SYSTEM Demo
  (* Version 1.0, 2022-05-14, Maximilian Scharf *)
  APPLICATION DemoApp
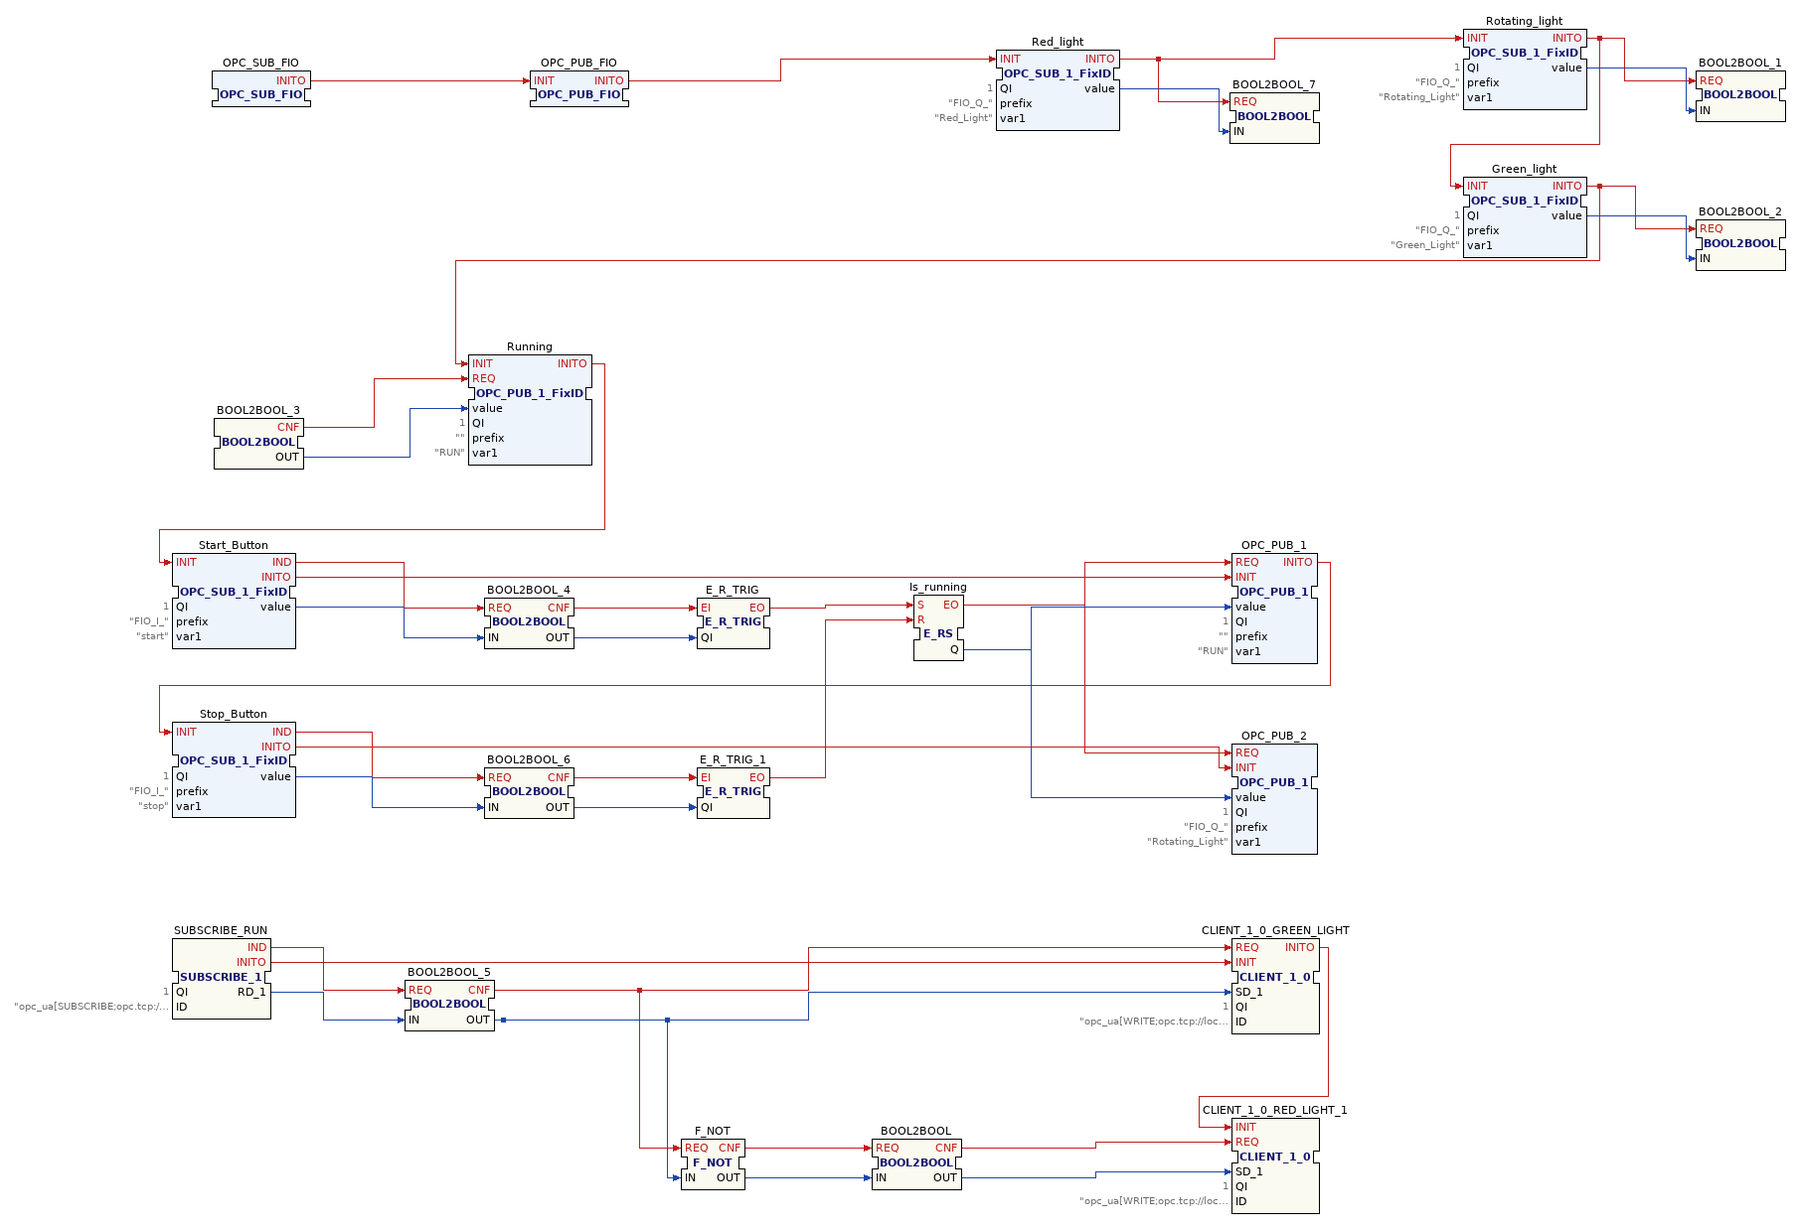
    (* Group __Group01: Factory IO controlpanel *)
    (* Group __Group02: Create nodes on server, which are used on clients *)
    (* Group __Group03: node RUN only writeable for server-forte *)
    FBS
      BOOL2BOOL_1 : BOOL2BOOL; {SET_ATTRIBUTE(GroupName, __Group02)}
      BOOL2BOOL_2 : BOOL2BOOL; {SET_ATTRIBUTE(GroupName, __Group02)}
      BOOL2BOOL_4 : BOOL2BOOL;
      Is_running : E_RS;
      BOOL2BOOL_5 : BOOL2BOOL;
      SUBSCRIBE_RUN : SUBSCRIBE_1(QI := 1, ID := "opc_ua[SUBSCRIBE;opc.tcp://localhost:4840#;/Objects/RUN]");
      CLIENT_1_0_GREEN_LIGHT : CLIENT_1_0(QI := 1, ID := "opc_ua[WRITE;opc.tcp://localhost:4840#;/Objects/FIO_Q_Green_Light]");
      BOOL2BOOL_3 : BOOL2BOOL; {SET_ATTRIBUTE(GroupName, __Group03)}
      E_R_TRIG : E_R_TRIG;
      E_R_TRIG_1 : E_R_TRIG;
      BOOL2BOOL_6 : BOOL2BOOL;
      BOOL2BOOL_7 : BOOL2BOOL; {SET_ATTRIBUTE(GroupName, __Group02)}
      F_NOT : F_NOT;
      CLIENT_1_0_RED_LIGHT_1 : CLIENT_1_0(QI := 1, ID := "opc_ua[WRITE;opc.tcp://localhost:4840#;/Objects/FIO_Q_Red_Light]");
      BOOL2BOOL : BOOL2BOOL;
    END_FBS
    SUBAPPS
      OPC_PUB_FIO : OPC_PUB_FIO; {SET_ATTRIBUTE(GroupName, __Group01)}
      Start_Button : OPC_SUB_1_FixID(QI := 1, prefix := "FIO_I_", var1 := "start");
      Rotating_light : OPC_SUB_1_FixID(QI := 1, prefix := "FIO_Q_", var1 := "Rotating_Light"); {SET_ATTRIBUTE(GroupName, __Group02)}
      Green_light : OPC_SUB_1_FixID(QI := 1, prefix := "FIO_Q_", var1 := "Green_Light"); {SET_ATTRIBUTE(GroupName, __Group02)}
      OPC_SUB_FIO : OPC_SUB_FIO; {SET_ATTRIBUTE(GroupName, __Group01)}
      OPC_PUB_1 : OPC_PUB_1(QI := 1, prefix := "", var1 := "RUN");
      OPC_PUB_2 : OPC_PUB_1(QI := 1, prefix := "FIO_Q_", var1 := "Rotating_Light");
      Running : OPC_PUB_1_FixID(QI := 1, prefix := "", var1 := "RUN"); {SET_ATTRIBUTE(GroupName, __Group03)}
      Stop_Button : OPC_SUB_1_FixID(QI := 1, prefix := "FIO_I_", var1 := "stop");
      Red_light : OPC_SUB_1_FixID(QI := 1, prefix := "FIO_Q_", var1 := "Red_Light"); {SET_ATTRIBUTE(GroupName, __Group02)}
    END_SUBAPPS
    EVENT_CONNECTIONS
      OPC_SUB_FIO.INITO TO OPC_PUB_FIO.INIT;
      Rotating_light.INITO TO BOOL2BOOL_1.REQ;
      Green_light.INITO TO BOOL2BOOL_2.REQ;
      Is_running.EO TO OPC_PUB_1.REQ;
      SUBSCRIBE_RUN.IND TO BOOL2BOOL_5.REQ;
      BOOL2BOOL_5.CNF TO CLIENT_1_0_GREEN_LIGHT.REQ;
      Green_light.INITO TO Running.INIT;
      BOOL2BOOL_3.CNF TO Running.REQ;
      Start_Button.IND TO BOOL2BOOL_4.REQ;
      Start_Button.INITO TO OPC_PUB_1.INIT;
      Running.INITO TO Start_Button.INIT;
      BOOL2BOOL_4.CNF TO E_R_TRIG.EI;
      E_R_TRIG.EO TO Is_running.S;
      Is_running.EO TO OPC_PUB_2.REQ;
      SUBSCRIBE_RUN.INITO TO CLIENT_1_0_GREEN_LIGHT.INIT;
      BOOL2BOOL_6.CNF TO E_R_TRIG_1.EI;
      Stop_Button.IND TO BOOL2BOOL_6.REQ;
      E_R_TRIG_1.EO TO Is_running.R;
      Red_light.INITO TO BOOL2BOOL_7.REQ;
      OPC_PUB_FIO.INITO TO Red_light.INIT;
      Red_light.INITO TO Rotating_light.INIT;
      OPC_PUB_1.INITO TO Stop_Button.INIT;
      Stop_Button.INITO TO OPC_PUB_2.INIT;
      BOOL2BOOL_5.CNF TO F_NOT.REQ;
      CLIENT_1_0_GREEN_LIGHT.INITO TO CLIENT_1_0_RED_LIGHT_1.INIT;
      F_NOT.CNF TO BOOL2BOOL.REQ;
      BOOL2BOOL.CNF TO CLIENT_1_0_RED_LIGHT_1.REQ;
      Rotating_light.INITO TO Green_light.INIT;
    END_CONNECTIONS
    DATA_CONNECTIONS
      Rotating_light.value TO BOOL2BOOL_1.IN;
      Green_light.value TO BOOL2BOOL_2.IN;
      Is_running.Q TO OPC_PUB_1.value;
      Is_running.Q TO OPC_PUB_2.value;
      SUBSCRIBE_RUN.RD_1 TO BOOL2BOOL_5.IN;
      BOOL2BOOL_5.OUT TO CLIENT_1_0_GREEN_LIGHT.SD_1;
      BOOL2BOOL_3.OUT TO Running.value;
      Start_Button.value TO BOOL2BOOL_4.IN;
      BOOL2BOOL_4.OUT TO E_R_TRIG.QI;
      Stop_Button.value TO BOOL2BOOL_6.IN;
      BOOL2BOOL_6.OUT TO E_R_TRIG_1.QI;
      Red_light.value TO BOOL2BOOL_7.IN;
      BOOL2BOOL_5.OUT TO F_NOT.IN;
      F_NOT.OUT TO BOOL2BOOL.IN;
      BOOL2BOOL.OUT TO CLIENT_1_0_RED_LIGHT_1.SD_1;
    END_CONNECTIONS
  END_APPLICATION
  DEVICE Server : FORTE_PC(MGR_ID := "localhost:61499")
    {SET_ATTRIBUTE(Profile, DynamicTypeLoad)}
    {SET_ATTRIBUTE(FBType, GEN_E_MUX, F_LT, F_LWORD_TO_WORD, F_TAN, F_DINT_TO_UINT, F_BYTE_TO_DINT, F_ADD_DT_TIME, F_TIME_IN_US_TO_LREAL, F_INT_TO_UDINT, F_ADD_TOD_TIME, F_SUB_DT_DT, F_DT_TO_TOD, F_WSTRING_TO_REAL, F_UINT_TO_BCD_WORD, F_UDINT_TO_REAL, F_REAL_TO_UDINT, F_DWORD_TO_WORD, F_MUL, FB_CTUD_LINT, TEST_CONDITION, F_LE, GEN_SUBSCRIBE, F_LN, FB_CTD_DINT, GEN_OR, E_CYCLE, FB_F_TRIG, F_LREAL_TO_SINT, E_F_TRIG, F_LWORD_TO_UINT, E_RS, F_UINT_TO_WORD, F_WORD_TO_DINT, F_OR, F_WORD_TO_BYTE, F_TIME_IN_NS_TO_ULINT, FB_CTD_ULINT, FB_TOF, STEST_END, F_NE, FB_TON, F_STRING_TO_UINT, F_LWORD_TO_ULINT, F_INT_TO_STRING, F_INT_TO_BYTE, F_INT_TO_DINT, F_ULINT_TO_LINT, F_DWORD_TO_UINT, F_WSTRING_TO_ULINT, F_WSTRING_TO_LWORD, F_STRING_TO_DWORD, DWORD2DWORD, F_TIME_IN_NS_TO_LINT, F_DINT_TO_WSTRING, E_SELECT, F_LINT_TO_STRING, FB_CTUD, F_MULTIME, F_USINT_TO_INT, LocalizedText2LocalizedText, F_DWORD_TO_UDINT, F_UINT_TO_LWORD, F_SINT_TO_LWORD, GEN_F_MUX, USINT2USINT, F_LINT_TO_SINT, F_WORD_TO_USINT, F_DWORD_TO_INT, F_LREAL_TO_REAL, F_BOOL_TO_LINT, F_LEFT, FB_CTD, E_SR, F_UDINT_TO_BCD_DWORD, GEN_XOR, F_DINT_TO_WORD, F_SUB_TOD_TIME, E_RESTART, E_PERMIT, TIME2TIME, F_UINT_TO_SINT, F_XOR, F_STRING_TO_WORD, F_SEL, F_ULINT_TO_LREAL, F_SINT_TO_LREAL, F_DINT_TO_SINT, E_TimeOut, F_BYTE_TO_UDINT, F_REPLACE, F_LINT_TO_USINT, F_ABS, F_WORD_TO_LWORD, E_DELAY, GEN_ADD, F_INT_TO_WSTRING, F_STRING_TO_ULINT, F_USINT_TO_STRING, F_DINT_TO_USINT, F_STRING_TO_BOOL, F_DWORD_TO_WSTRING, F_INT_TO_REAL, F_DWORD_TO_STRING, E_CTU, F_TIME_TO_STRING, F_WSTRING_TO_BYTE, F_USINT_TO_WSTRING, F_WSTRING_TO_DINT, F_WSTRING_TO_DWORD, F_MOVE, F_WSTRING_TO_STRING, F_USINT_TO_LINT, F_DIV, F_WSTRING_TO_SINT, E_CTD, F_UINT_TO_DWORD, F_LWORD_TO_LINT, F_STRING_TO_TIME, FB_CTUD_DINT, F_ADD, F_BYTE_TO_LINT, F_TIME_IN_MS_TO_LREAL, F_LREAL_TO_UINT, F_ACOS, F_DWORD_TO_LINT, F_SHL, F_REAL_TO_ULINT, F_ULINT_TO_UINT, F_UDINT_TO_SINT, F_SHR, F_BOOL_TO_INT, UINT2UINT, F_WORD_TO_DWORD, F_INT_TO_LWORD, F_USINT_TO_UINT, F_LREAL_TO_WSTRING, F_INT_TO_ULINT, GEN_CSV_WRITER, F_LINT_TO_WORD, F_UINT_TO_LREAL, F_STRING_TO_SINT, F_SINT_TO_WORD, F_STRING_TO_WSTRING, STRING2STRING, F_LREAL_TO_DINT, F_SIN, F_UINT_TO_USINT, FB_CTU_LINT, F_DINT_TO_ULINT, F_REAL_TO_UINT, RMT_RES, F_ULINT_TO_WORD, F_INT_TO_LINT, E_D_FF, F_STRING_TO_USINT, FB_CTD_LINT, FB_R_TRIG, F_INT_TO_DWORD, F_WORD_TO_LINT, F_UDINT_TO_INT, REAL2REAL, F_LREAL_TO_STRING, F_WSTRING_TO_INT, F_LREAL_TO_USINT, F_DINT_TO_LWORD, DEV_MGR, F_SINT_TO_UINT, E_CTUD, E_RDELAY, F_SINT_TO_ULINT, F_LINT_TO_ULINT, F_RIGHT, F_SINT_TO_INT, F_LWORD_TO_WSTRING, SINT2SINT, FB_CTD_UDINT, F_LINT_TO_LWORD, F_LWORD_TO_UDINT, F_LWORD_TO_STRING, F_TRUNC, F_ULINT_TO_DWORD, F_TIME_IN_S_TO_LREAL, F_BOOL_TO_DWORD, E_TRAIN, OUT_ANY_CONSOLE, F_ULINT_TO_SINT, F_DINT_TO_LINT, F_BOOL_TO_USINT, F_UDINT_TO_DWORD, GEN_E_DEMUX, F_SQRT, F_BOOL_TO_DINT, F_BOOL_TO_BYTE, F_UINT_TO_INT, F_TIME_IN_S_TO_LINT, F_ULINT_TO_USINT, F_UINT_TO_REAL, F_LREAL_TO_LWORD, F_SINT_TO_LINT, F_MAX, F_LREAL_TO_INT, F_UDINT_TO_LWORD, INT2INT, F_BYTE_TO_ULINT, F_UDINT_TO_WORD, F_LINT_TO_UINT, F_TIME_IN_US_TO_ULINT, F_COS, F_TIME_IN_NS_TO_LREAL, F_REAL_TO_LINT, F_STRING_TO_LWORD, F_BYTE_TO_STRING, F_USINT_TO_WORD, E_REND, F_ASIN, F_REAL_TO_INT, F_BOOL_TO_LWORD, F_WORD_BCD_TO_UINT, F_BOOL_TO_SINT, F_BYTE_TO_INT, F_BOOL_TO_ULINT, EMB_RES, F_BYTE_TO_WORD, F_STRING_TO_INT, F_USINT_TO_LWORD, F_DWORD_TO_DINT, F_ULINT_TO_LWORD, GEN_APPEND_STRING, F_USINT_TO_ULINT, GEN_SUBL, F_DWORD_TO_BYTE, F_DIVTIME, F_ROL, F_LWORD_TO_DINT, F_WORD_TO_SINT, F_STRING_TO_REAL, F_LWORD_TO_BYTE, FB_CTU_DINT, GEN_AND, F_AND, F_ROR, GEN_CLIENT, F_ULINT_TO_WSTRING, F_SINT_TO_STRING, F_LREAL_TO_LINT, WSTRING2WSTRING, F_WORD_TO_INT, F_UINT_TO_BYTE, F_UDINT_TO_UINT, F_SINT_TO_UDINT, F_UINT_TO_DINT, F_UINT_TO_UDINT, F_UINT_TO_WSTRING, F_WSTRING_TO_UINT, F_DINT_TO_UDINT, E_SPLIT, F_DWORD_TO_LWORD, F_USINT_TO_SINT, F_ULINT_TO_BCD_LWORD, F_BYTE_BCD_TO_USINT, F_DWORD_TO_ULINT, F_BYTE_TO_SINT, F_BYTE_TO_WSTRING, GEN_ARRAY2ARRAY, F_DT_TO_DATE, GEN_STRUCT_DEMUX, F_LEN, GEN_STRUCT_MUX, F_INT_TO_WORD, FB_RANDOM, F_LINT_TO_UDINT, F_EXP, F_USINT_TO_DWORD, F_TIME_IN_MS_TO_ULINT, F_REAL_TO_SINT, F_INT_TO_USINT, F_UDINT_TO_WSTRING, F_EXPT, F_SUB, F_ULINT_TO_REAL, F_REAL_TO_LREAL, F_MID, F_BYTE_TO_UINT, F_BYTE_TO_DWORD, F_INT_TO_UINT, F_DWORD_TO_REAL, F_DINT_TO_BYTE, F_WORD_TO_STRING, F_REAL_TO_STRING, F_SUB_TOD_TOD, SET_AT_INDEX, F_MIN, F_LREAL_TO_ULINT, F_STRING_TO_BYTE, F_BYTE_TO_LWORD, F_STRING_TO_DINT, F_WORD_TO_WSTRING, BOOL2BOOL, F_LINT_TO_INT, F_WSTRING_TO_TIME, FB_CTU_UDINT, F_WSTRING_TO_BOOL, F_INSERT, F_SUB_DT_TIME, F_FIND, F_UDINT_TO_ULINT, F_WORD_TO_UDINT, F_DINT_TO_DWORD, F_WSTRING_TO_USINT, GEN_VALUES2ARRAY, GEN_ARRAY2VALUES, F_WSTRING_TO_WORD, F_DINT_TO_STRING, F_WORD_TO_UINT, F_TIME_IN_US_TO_LINT, F_LINT_TO_DWORD, F_CONCAT, FB_CTUD_ULINT, F_UDINT_TO_LINT, F_SUB_DATE_DATE, F_LWORD_TO_LREAL, F_LWORD_TO_INT, WORD2WORD, E_STOPWATCH, F_LIMIT, F_TIME_IN_S_TO_ULINT, F_LWORD_TO_USINT, F_REAL_TO_DINT, F_DWORD_TO_USINT, E_MERGE, F_SINT_TO_DWORD, E_DEMUX, F_BOOL_TO_UDINT, BYTE2BYTE, FB_TP, F_USINT_TO_BCD_BYTE, F_SINT_TO_DINT, F_UINT_TO_LINT, F_SINT_TO_BYTE, F_ATAN, F_LINT_TO_BYTE, F_BYTE_TO_USINT, F_ULINT_TO_UDINT, FB_SR, F_NOT, F_DINT_TO_INT, F_LINT_TO_DINT, F_DELETE, FB_CTU, GEN_SERVER, GEN_PUBL, F_UDINT_TO_LREAL, F_BOOL_TO_UINT, F_UINT_TO_STRING, E_R_TRIG, F_GE, F_LWORD_BCD_TO_ULINT, F_UDINT_TO_STRING, F_REAL_TO_WSTRING, FB_RS, F_MUX_2, F_LINT_TO_WSTRING, F_USINT_TO_UDINT, F_UINT_TO_ULINT, F_EQ, E_T_FF, F_USINT_TO_REAL, LREAL2LREAL, F_STRING_TO_LREAL, F_ULINT_TO_STRING, F_MOD, E_RTimeOut, F_ULINT_TO_DINT, F_ULINT_TO_BYTE, F_WSTRING_TO_UDINT, F_TIME_TO_WSTRING, GET_STRUCT_VALUE, GEN_PUBLISH, F_REAL_TO_DWORD, F_DWORD_BCD_TO_UDINT, F_INT_TO_LREAL, F_SINT_TO_WSTRING, F_LWORD_TO_SINT, F_GT, F_LINT_TO_REAL, F_TIME_IN_MS_TO_LINT, F_SINT_TO_REAL, F_LOG, F_ULINT_TO_INT, F_DWORD_TO_SINT, F_BOOL_TO_WORD, F_REAL_TO_USINT, E_SWITCH, F_LINT_TO_LREAL, F_STRING_TO_LINT, F_SINT_TO_USINT, F_DINT_TO_REAL, DINT2DINT, F_WORD_TO_ULINT, F_INT_TO_SINT, F_CONCAT_DATE_TOD, F_WSTRING_TO_LREAL, GET_AT_INDEX, F_USINT_TO_LREAL, F_BOOL_TO_WSTRING, FB_CTU_ULINT, F_DINT_TO_LREAL, UDINT2UDINT, F_USINT_TO_BYTE, F_BOOL_TO_STRING, F_LWORD_TO_DWORD, F_LREAL_TO_UDINT, F_STRING_TO_UDINT, F_UDINT_TO_DINT, F_UDINT_TO_BYTE, F_WSTRING_TO_LINT, F_USINT_TO_DINT)} (* created during deployment *)
    RESOURCE EMB_RES : EMB_RES
      FBS
        BOOL2BOOL_7 : BOOL2BOOL;
        BOOL2BOOL_6 : BOOL2BOOL;
        E_R_TRIG_1 : E_R_TRIG;
        E_R_TRIG : E_R_TRIG;
        BOOL2BOOL_3 : BOOL2BOOL;
        Is_running : E_RS;
        BOOL2BOOL_4 : BOOL2BOOL;
        BOOL2BOOL_2 : BOOL2BOOL;
        BOOL2BOOL_1 : BOOL2BOOL;
      END_FBS
      SUBAPPS
        Red_light : OPC_SUB_1_FixID(QI := 1, prefix := "FIO_Q_", var1 := "Red_Light");
        Stop_Button : OPC_SUB_1_FixID(QI := 1, prefix := "FIO_I_", var1 := "stop");
        Running : OPC_PUB_1_FixID(QI := 1, prefix := "", var1 := "RUN");
        OPC_PUB_2 : OPC_PUB_1(QI := 1, prefix := "FIO_Q_", var1 := "Rotating_Light");
        OPC_PUB_1 : OPC_PUB_1(QI := 1, prefix := "", var1 := "RUN");
        OPC_SUB_FIO : OPC_SUB_FIO;
        Green_light : OPC_SUB_1_FixID(QI := 1, prefix := "FIO_Q_", var1 := "Green_Light");
        Rotating_light : OPC_SUB_1_FixID(QI := 1, prefix := "FIO_Q_", var1 := "Rotating_Light");
        Start_Button : OPC_SUB_1_FixID(QI := 1, prefix := "FIO_I_", var1 := "start");
        OPC_PUB_FIO : OPC_PUB_FIO;
      END_SUBAPPS
      EVENT_CONNECTIONS
        Red_light.INITO TO BOOL2BOOL_7.REQ;
        Stop_Button.IND TO BOOL2BOOL_6.REQ;
        BOOL2BOOL_6.CNF TO E_R_TRIG_1.EI;
        BOOL2BOOL_3.CNF TO Running.REQ;
        Stop_Button.INITO TO OPC_PUB_2.INIT;
        OPC_PUB_1.INITO TO Stop_Button.INIT;
        Is_running.EO TO OPC_PUB_2.REQ;
        Is_running.EO TO OPC_PUB_1.REQ;
        E_R_TRIG.EO TO Is_running.S;
        E_R_TRIG_1.EO TO Is_running.R;
        BOOL2BOOL_4.CNF TO E_R_TRIG.EI;
        START.COLD TO OPC_SUB_FIO.INIT;
        Green_light.INITO TO BOOL2BOOL_2.REQ;
        Green_light.INITO TO Running.INIT;
        Rotating_light.INITO TO BOOL2BOOL_1.REQ;
        Red_light.INITO TO Rotating_light.INIT;
        Start_Button.IND TO BOOL2BOOL_4.REQ;
        Start_Button.INITO TO OPC_PUB_1.INIT;
        Running.INITO TO Start_Button.INIT;
        OPC_PUB_FIO.INITO TO Red_light.INIT;
        OPC_SUB_FIO.INITO TO OPC_PUB_FIO.INIT;
        Rotating_light.INITO TO Green_light.INIT;
      END_CONNECTIONS
      DATA_CONNECTIONS
        Red_light.value TO BOOL2BOOL_7.IN;
        Stop_Button.value TO BOOL2BOOL_6.IN;
        BOOL2BOOL_6.OUT TO E_R_TRIG_1.QI;
        BOOL2BOOL_3.OUT TO Running.value;
        Is_running.Q TO OPC_PUB_1.value;
        Is_running.Q TO OPC_PUB_2.value;
        BOOL2BOOL_4.OUT TO E_R_TRIG.QI;
        Green_light.value TO BOOL2BOOL_2.IN;
        Rotating_light.value TO BOOL2BOOL_1.IN;
        Start_Button.value TO BOOL2BOOL_4.IN;
      END_CONNECTIONS
    END_RESOURCE
  END_DEVICE
  DEVICE Client : FORTE_PC(MGR_ID := "localhost:61599")
    {SET_ATTRIBUTE(Profile, DynamicTypeLoad)}
    {SET_ATTRIBUTE(FBType, GEN_E_MUX, F_LT, F_LWORD_TO_WORD, F_TAN, F_DINT_TO_UINT, F_BYTE_TO_DINT, F_ADD_DT_TIME, F_TIME_IN_US_TO_LREAL, F_INT_TO_UDINT, F_ADD_TOD_TIME, F_SUB_DT_DT, F_DT_TO_TOD, F_WSTRING_TO_REAL, F_UINT_TO_BCD_WORD, F_UDINT_TO_REAL, F_REAL_TO_UDINT, F_DWORD_TO_WORD, F_MUL, FB_CTUD_LINT, TEST_CONDITION, F_LE, GEN_SUBSCRIBE, F_LN, FB_CTD_DINT, GEN_OR, E_CYCLE, FB_F_TRIG, F_LREAL_TO_SINT, E_F_TRIG, F_LWORD_TO_UINT, E_RS, F_UINT_TO_WORD, F_WORD_TO_DINT, F_OR, F_WORD_TO_BYTE, F_TIME_IN_NS_TO_ULINT, FB_CTD_ULINT, FB_TOF, STEST_END, F_NE, FB_TON, F_STRING_TO_UINT, F_LWORD_TO_ULINT, F_INT_TO_STRING, F_INT_TO_BYTE, F_INT_TO_DINT, F_ULINT_TO_LINT, F_DWORD_TO_UINT, F_WSTRING_TO_ULINT, F_WSTRING_TO_LWORD, F_STRING_TO_DWORD, DWORD2DWORD, F_TIME_IN_NS_TO_LINT, F_DINT_TO_WSTRING, E_SELECT, F_LINT_TO_STRING, FB_CTUD, F_MULTIME, F_USINT_TO_INT, LocalizedText2LocalizedText, F_DWORD_TO_UDINT, F_UINT_TO_LWORD, F_SINT_TO_LWORD, GEN_F_MUX, USINT2USINT, F_LINT_TO_SINT, F_WORD_TO_USINT, F_DWORD_TO_INT, F_LREAL_TO_REAL, F_BOOL_TO_LINT, F_LEFT, FB_CTD, E_SR, F_UDINT_TO_BCD_DWORD, GEN_XOR, F_DINT_TO_WORD, F_SUB_TOD_TIME, E_RESTART, E_PERMIT, TIME2TIME, F_UINT_TO_SINT, F_XOR, F_STRING_TO_WORD, F_SEL, F_ULINT_TO_LREAL, F_SINT_TO_LREAL, F_DINT_TO_SINT, E_TimeOut, F_BYTE_TO_UDINT, F_REPLACE, F_LINT_TO_USINT, F_ABS, F_WORD_TO_LWORD, E_DELAY, GEN_ADD, F_INT_TO_WSTRING, F_STRING_TO_ULINT, F_USINT_TO_STRING, F_DINT_TO_USINT, F_STRING_TO_BOOL, F_DWORD_TO_WSTRING, F_INT_TO_REAL, F_DWORD_TO_STRING, E_CTU, F_TIME_TO_STRING, F_WSTRING_TO_BYTE, F_USINT_TO_WSTRING, F_WSTRING_TO_DINT, F_WSTRING_TO_DWORD, F_MOVE, F_WSTRING_TO_STRING, F_USINT_TO_LINT, F_DIV, F_WSTRING_TO_SINT, E_CTD, F_UINT_TO_DWORD, F_LWORD_TO_LINT, F_STRING_TO_TIME, FB_CTUD_DINT, F_ADD, F_BYTE_TO_LINT, F_TIME_IN_MS_TO_LREAL, F_LREAL_TO_UINT, F_ACOS, F_DWORD_TO_LINT, F_SHL, F_REAL_TO_ULINT, F_ULINT_TO_UINT, F_UDINT_TO_SINT, F_SHR, F_BOOL_TO_INT, UINT2UINT, F_WORD_TO_DWORD, F_INT_TO_LWORD, F_USINT_TO_UINT, F_LREAL_TO_WSTRING, F_INT_TO_ULINT, GEN_CSV_WRITER, F_LINT_TO_WORD, F_UINT_TO_LREAL, F_STRING_TO_SINT, F_SINT_TO_WORD, F_STRING_TO_WSTRING, STRING2STRING, F_LREAL_TO_DINT, F_SIN, F_UINT_TO_USINT, FB_CTU_LINT, F_DINT_TO_ULINT, F_REAL_TO_UINT, RMT_RES, F_ULINT_TO_WORD, F_INT_TO_LINT, E_D_FF, F_STRING_TO_USINT, FB_CTD_LINT, FB_R_TRIG, F_INT_TO_DWORD, F_WORD_TO_LINT, F_UDINT_TO_INT, REAL2REAL, F_LREAL_TO_STRING, F_WSTRING_TO_INT, F_LREAL_TO_USINT, F_DINT_TO_LWORD, DEV_MGR, F_SINT_TO_UINT, E_CTUD, E_RDELAY, F_SINT_TO_ULINT, F_LINT_TO_ULINT, F_RIGHT, F_SINT_TO_INT, F_LWORD_TO_WSTRING, SINT2SINT, FB_CTD_UDINT, F_LINT_TO_LWORD, F_LWORD_TO_UDINT, F_LWORD_TO_STRING, F_TRUNC, F_ULINT_TO_DWORD, F_TIME_IN_S_TO_LREAL, F_BOOL_TO_DWORD, E_TRAIN, OUT_ANY_CONSOLE, F_ULINT_TO_SINT, F_DINT_TO_LINT, F_BOOL_TO_USINT, F_UDINT_TO_DWORD, GEN_E_DEMUX, F_SQRT, F_BOOL_TO_DINT, F_BOOL_TO_BYTE, F_UINT_TO_INT, F_TIME_IN_S_TO_LINT, F_ULINT_TO_USINT, F_UINT_TO_REAL, F_LREAL_TO_LWORD, F_SINT_TO_LINT, F_MAX, F_LREAL_TO_INT, F_UDINT_TO_LWORD, INT2INT, F_BYTE_TO_ULINT, F_UDINT_TO_WORD, F_LINT_TO_UINT, F_TIME_IN_US_TO_ULINT, F_COS, F_TIME_IN_NS_TO_LREAL, F_REAL_TO_LINT, F_STRING_TO_LWORD, F_BYTE_TO_STRING, F_USINT_TO_WORD, E_REND, F_ASIN, F_REAL_TO_INT, F_BOOL_TO_LWORD, F_WORD_BCD_TO_UINT, F_BOOL_TO_SINT, F_BYTE_TO_INT, F_BOOL_TO_ULINT, EMB_RES, F_BYTE_TO_WORD, F_STRING_TO_INT, F_USINT_TO_LWORD, F_DWORD_TO_DINT, F_ULINT_TO_LWORD, GEN_APPEND_STRING, F_USINT_TO_ULINT, GEN_SUBL, F_DWORD_TO_BYTE, F_DIVTIME, F_ROL, F_LWORD_TO_DINT, F_WORD_TO_SINT, F_STRING_TO_REAL, F_LWORD_TO_BYTE, FB_CTU_DINT, GEN_AND, F_AND, F_ROR, GEN_CLIENT, F_ULINT_TO_WSTRING, F_SINT_TO_STRING, F_LREAL_TO_LINT, WSTRING2WSTRING, F_WORD_TO_INT, F_UINT_TO_BYTE, F_UDINT_TO_UINT, F_SINT_TO_UDINT, F_UINT_TO_DINT, F_UINT_TO_UDINT, F_UINT_TO_WSTRING, F_WSTRING_TO_UINT, F_DINT_TO_UDINT, E_SPLIT, F_DWORD_TO_LWORD, F_USINT_TO_SINT, F_ULINT_TO_BCD_LWORD, F_BYTE_BCD_TO_USINT, F_DWORD_TO_ULINT, F_BYTE_TO_SINT, F_BYTE_TO_WSTRING, GEN_ARRAY2ARRAY, F_DT_TO_DATE, GEN_STRUCT_DEMUX, F_LEN, GEN_STRUCT_MUX, F_INT_TO_WORD, FB_RANDOM, F_LINT_TO_UDINT, F_EXP, F_USINT_TO_DWORD, F_TIME_IN_MS_TO_ULINT, F_REAL_TO_SINT, F_INT_TO_USINT, F_UDINT_TO_WSTRING, F_EXPT, F_SUB, F_ULINT_TO_REAL, F_REAL_TO_LREAL, F_MID, F_BYTE_TO_UINT, F_BYTE_TO_DWORD, F_INT_TO_UINT, F_DWORD_TO_REAL, F_DINT_TO_BYTE, F_WORD_TO_STRING, F_REAL_TO_STRING, F_SUB_TOD_TOD, SET_AT_INDEX, F_MIN, F_LREAL_TO_ULINT, F_STRING_TO_BYTE, F_BYTE_TO_LWORD, F_STRING_TO_DINT, F_WORD_TO_WSTRING, BOOL2BOOL, F_LINT_TO_INT, F_WSTRING_TO_TIME, FB_CTU_UDINT, F_WSTRING_TO_BOOL, F_INSERT, F_SUB_DT_TIME, F_FIND, F_UDINT_TO_ULINT, F_WORD_TO_UDINT, F_DINT_TO_DWORD, F_WSTRING_TO_USINT, GEN_VALUES2ARRAY, GEN_ARRAY2VALUES, F_WSTRING_TO_WORD, F_DINT_TO_STRING, F_WORD_TO_UINT, F_TIME_IN_US_TO_LINT, F_LINT_TO_DWORD, F_CONCAT, FB_CTUD_ULINT, F_UDINT_TO_LINT, F_SUB_DATE_DATE, F_LWORD_TO_LREAL, F_LWORD_TO_INT, WORD2WORD, E_STOPWATCH, F_LIMIT, F_TIME_IN_S_TO_ULINT, F_LWORD_TO_USINT, F_REAL_TO_DINT, F_DWORD_TO_USINT, E_MERGE, F_SINT_TO_DWORD, E_DEMUX, F_BOOL_TO_UDINT, BYTE2BYTE, FB_TP, F_USINT_TO_BCD_BYTE, F_SINT_TO_DINT, F_UINT_TO_LINT, F_SINT_TO_BYTE, F_ATAN, F_LINT_TO_BYTE, F_BYTE_TO_USINT, F_ULINT_TO_UDINT, FB_SR, F_NOT, F_DINT_TO_INT, F_LINT_TO_DINT, F_DELETE, FB_CTU, GEN_SERVER, GEN_PUBL, F_UDINT_TO_LREAL, F_BOOL_TO_UINT, F_UINT_TO_STRING, E_R_TRIG, F_GE, F_LWORD_BCD_TO_ULINT, F_UDINT_TO_STRING, F_REAL_TO_WSTRING, FB_RS, F_MUX_2, F_LINT_TO_WSTRING, F_USINT_TO_UDINT, F_UINT_TO_ULINT, F_EQ, E_T_FF, F_USINT_TO_REAL, LREAL2LREAL, F_STRING_TO_LREAL, F_ULINT_TO_STRING, F_MOD, E_RTimeOut, F_ULINT_TO_DINT, F_ULINT_TO_BYTE, F_WSTRING_TO_UDINT, F_TIME_TO_WSTRING, GET_STRUCT_VALUE, GEN_PUBLISH, F_REAL_TO_DWORD, F_DWORD_BCD_TO_UDINT, F_INT_TO_LREAL, F_SINT_TO_WSTRING, F_LWORD_TO_SINT, F_GT, F_LINT_TO_REAL, F_TIME_IN_MS_TO_LINT, F_SINT_TO_REAL, F_LOG, F_ULINT_TO_INT, F_DWORD_TO_SINT, F_BOOL_TO_WORD, F_REAL_TO_USINT, E_SWITCH, F_LINT_TO_LREAL, F_STRING_TO_LINT, F_SINT_TO_USINT, F_DINT_TO_REAL, DINT2DINT, F_WORD_TO_ULINT, F_INT_TO_SINT, F_CONCAT_DATE_TOD, F_WSTRING_TO_LREAL, GET_AT_INDEX, F_USINT_TO_LREAL, F_BOOL_TO_WSTRING, FB_CTU_ULINT, F_DINT_TO_LREAL, UDINT2UDINT, F_USINT_TO_BYTE, F_BOOL_TO_STRING, F_LWORD_TO_DWORD, F_LREAL_TO_UDINT, F_STRING_TO_UDINT, F_UDINT_TO_DINT, F_UDINT_TO_BYTE, F_WSTRING_TO_LINT, F_USINT_TO_DINT)} (* created during deployment *)
    RESOURCE EMB_RES : EMB_RES
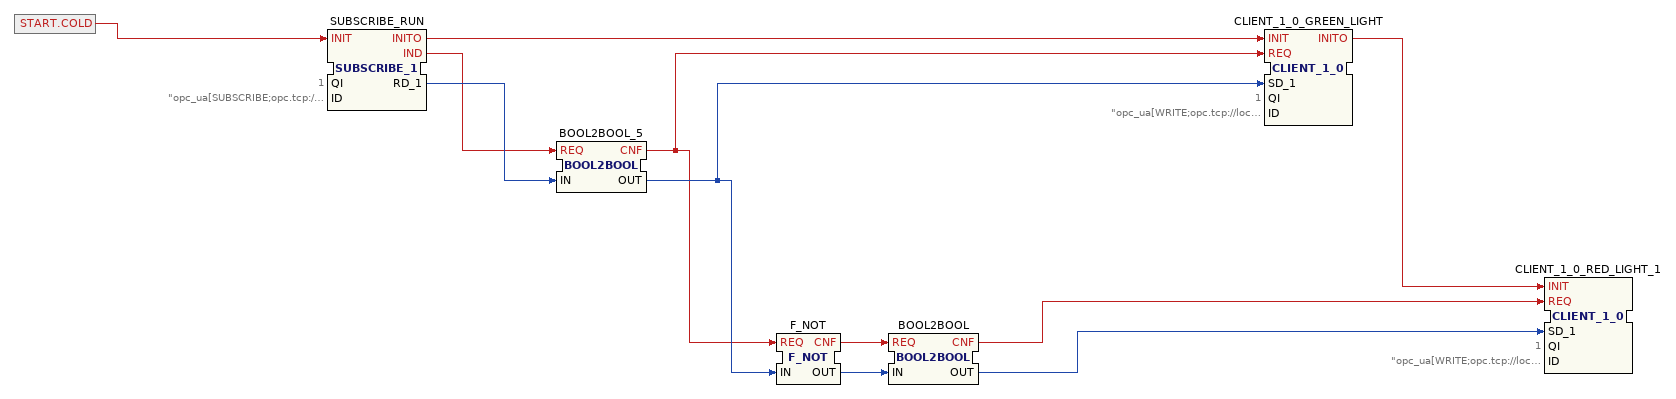
      FBS
        CLIENT_1_0_GREEN_LIGHT : CLIENT_1_0(QI := 1, ID := "opc_ua[WRITE;opc.tcp://localhost:4840#;/Objects/FIO_Q_Green_Light]");
        SUBSCRIBE_RUN : SUBSCRIBE_1(QI := 1, ID := "opc_ua[SUBSCRIBE;opc.tcp://localhost:4840#;/Objects/RUN]");
        BOOL2BOOL_5 : BOOL2BOOL;
        CLIENT_1_0_RED_LIGHT_1 : CLIENT_1_0(QI := 1, ID := "opc_ua[WRITE;opc.tcp://localhost:4840#;/Objects/FIO_Q_Red_Light]");
        F_NOT : F_NOT;
        BOOL2BOOL : BOOL2BOOL;
      END_FBS
      EVENT_CONNECTIONS
        SUBSCRIBE_RUN.INITO TO CLIENT_1_0_GREEN_LIGHT.INIT;
        START.COLD TO SUBSCRIBE_RUN.INIT;
        BOOL2BOOL_5.CNF TO CLIENT_1_0_GREEN_LIGHT.REQ;
        SUBSCRIBE_RUN.IND TO BOOL2BOOL_5.REQ;
        BOOL2BOOL_5.CNF TO F_NOT.REQ;
        CLIENT_1_0_GREEN_LIGHT.INITO TO CLIENT_1_0_RED_LIGHT_1.INIT;
        F_NOT.CNF TO BOOL2BOOL.REQ;
        BOOL2BOOL.CNF TO CLIENT_1_0_RED_LIGHT_1.REQ;
      END_CONNECTIONS
      DATA_CONNECTIONS
        BOOL2BOOL_5.OUT TO CLIENT_1_0_GREEN_LIGHT.SD_1;
        SUBSCRIBE_RUN.RD_1 TO BOOL2BOOL_5.IN;
        BOOL2BOOL_5.OUT TO F_NOT.IN;
        F_NOT.OUT TO BOOL2BOOL.IN;
        BOOL2BOOL.OUT TO CLIENT_1_0_RED_LIGHT_1.SD_1;
      END_CONNECTIONS
    END_RESOURCE
  END_DEVICE
  MAPPINGS
    DemoApp.BOOL2BOOL_7 ON Server.EMB_RES.BOOL2BOOL_7;
    DemoApp.Red_light ON Server.EMB_RES.Red_light;
    DemoApp.Stop_Button ON Server.EMB_RES.Stop_Button;
    DemoApp.BOOL2BOOL_6 ON Server.EMB_RES.BOOL2BOOL_6;
    DemoApp.E_R_TRIG_1 ON Server.EMB_RES.E_R_TRIG_1;
    DemoApp.E_R_TRIG ON Server.EMB_RES.E_R_TRIG;
    DemoApp.BOOL2BOOL_3 ON Server.EMB_RES.BOOL2BOOL_3;
    DemoApp.Running ON Server.EMB_RES.Running;
    DemoApp.CLIENT_1_0_GREEN_LIGHT ON Client.EMB_RES.CLIENT_1_0_GREEN_LIGHT;
    DemoApp.SUBSCRIBE_RUN ON Client.EMB_RES.SUBSCRIBE_RUN;
    DemoApp.BOOL2BOOL_5 ON Client.EMB_RES.BOOL2BOOL_5;
    DemoApp.OPC_PUB_2 ON Server.EMB_RES.OPC_PUB_2;
    DemoApp.OPC_PUB_1 ON Server.EMB_RES.OPC_PUB_1;
    DemoApp.Is_running ON Server.EMB_RES.Is_running;
    DemoApp.BOOL2BOOL_4 ON Server.EMB_RES.BOOL2BOOL_4;
    DemoApp.BOOL2BOOL_2 ON Server.EMB_RES.BOOL2BOOL_2;
    DemoApp.BOOL2BOOL_1 ON Server.EMB_RES.BOOL2BOOL_1;
    DemoApp.OPC_SUB_FIO ON Server.EMB_RES.OPC_SUB_FIO;
    DemoApp.Green_light ON Server.EMB_RES.Green_light;
    DemoApp.Rotating_light ON Server.EMB_RES.Rotating_light;
    DemoApp.Start_Button ON Server.EMB_RES.Start_Button;
    DemoApp.OPC_PUB_FIO ON Server.EMB_RES.OPC_PUB_FIO;
    DemoApp.CLIENT_1_0_RED_LIGHT_1 ON Client.EMB_RES.CLIENT_1_0_RED_LIGHT_1;
    DemoApp.F_NOT ON Client.EMB_RES.F_NOT;
    DemoApp.BOOL2BOOL ON Client.EMB_RES.BOOL2BOOL;
  END_MAPPINGS
END_SYSTEM
